// TIA Portal V20 export
DATA_BLOCK "ProcessValues_DB"   // DB34
AUTHOR : Siemens AG
FAMILY : ServiceControl
VERSION : 1.0
// stored: InstanceOfName ProcessValues, InstanceOfType FB
"ProcessValues"
   // VAR_INPUT
   //    ProcessValueOutAnalogIn { ExternalAccessible := 'False'; ExternalVisible := 'False'; ExternalWritable := 'False'} : Array[0..0] of "UDT_MTP_AnaProcessValueOut";
   //    ProcessValueOutDigitalIn { ExternalAccessible := 'False'; ExternalVisible := 'False'; ExternalWritable := 'False'} : Array[0..0] of "UDT_MTP_DIntProcessValueOut";
   //    ProcessValueOutBinaryIn { ExternalAccessible := 'False'; ExternalVisible := 'False'; ExternalWritable := 'False'} : Array[0..0] of "UDT_MTP_BinProcessValueOut";
   //    ProcessValueOutStringIn { ExternalAccessible := 'False'; ExternalVisible := 'False'; ExternalWritable := 'False'} : Array[0..0] of "UDT_MTP_StringProcessValueOut";
   //    ProcessValueInAnalogApply { ExternalAccessible := 'False'; ExternalVisible := 'False'; ExternalWritable := 'False'} : Array[0..0] of "UDT_Service_ProcessValueInApply";
   //    ProcessValueInDigitalApply { ExternalAccessible := 'False'; ExternalVisible := 'False'; ExternalWritable := 'False'} : Array[0..0] of "UDT_Service_ProcessValueInApply";
   // END_VAR
   // VAR_OUTPUT
   //    ProcessValueInAnalogOut { ExternalAccessible := 'False'; ExternalVisible := 'False'; ExternalWritable := 'False'} : Array[0..0] of "UDT_MTP_AnaProcessValueOut";
   //    ProcessValueInDigitalOut { ExternalAccessible := 'False'; ExternalVisible := 'False'; ExternalWritable := 'False'} : Array[0..0] of "UDT_MTP_DIntProcessValueOut";
   //    ProcessValueInBinaryOut { ExternalAccessible := 'False'; ExternalVisible := 'False'; ExternalWritable := 'False'} : Array[0..0] of "UDT_MTP_BinProcessValueOut";
   //    ProcessValueInStringOut { ExternalAccessible := 'False'; ExternalVisible := 'False'; ExternalWritable := 'False'} : Array[0..0] of "UDT_MTP_StringProcessValueOut";
   // END_VAR
   // VAR
   //    MTPAnalogIn : Array[0..4] of "UDT_MTP_AnaProcessValueIn";
   //    MTPDigitalIn : Array[0..0] of "UDT_MTP_DIntProcessValueIn";
   //    MTPBinaryIn : Array[0..0] of "UDT_MTP_BinProcessValueIn";
   //    MTPStringIn : Array[0..0] of "UDT_MTP_StringProcessValueIn";
   //    AnalogIn { ExternalAccessible := 'False'; ExternalVisible := 'False'; ExternalWritable := 'False'; S7_SetPoint := 'True'} : Array[0..0] of "ProcessValueInAnalog";
   //    DigitalIn { ExternalAccessible := 'False'; ExternalVisible := 'False'; ExternalWritable := 'False'; S7_SetPoint := 'True'} : Array[0..0] of "ProcessValueInDigital";
   //    BinaryIn { ExternalAccessible := 'False'; ExternalVisible := 'False'; ExternalWritable := 'False'; S7_SetPoint := 'True'} : Array[0..0] of "ProcessValueInBinary";
   //    StringIn { ExternalAccessible := 'False'; ExternalVisible := 'False'; ExternalWritable := 'False'; S7_SetPoint := 'True'} : Array[0..0] of "ProcessValueInString";
   //    MTPAnalogOut : Array[0..10] of "UDT_MTP_AnaProcessValueOut";
   //    MTPDigitalOut : Array[0..0] of "UDT_MTP_DIntProcessValueOut";
   //    MTPBinaryOut : Array[0..2] of "UDT_MTP_BinProcessValueOut";
   //    MTPStringOut : Array[0..0] of "UDT_MTP_StringProcessValueOut";
   //    AnalogOut { ExternalAccessible := 'False'; ExternalVisible := 'False'; ExternalWritable := 'False'; S7_SetPoint := 'True'} : Array[0..0] of "ProcessValueOutAnalog";
   //    DigitalOut { ExternalAccessible := 'False'; ExternalVisible := 'False'; ExternalWritable := 'False'; S7_SetPoint := 'True'} : Array[0..0] of "ProcessValueOutDigital";
   //    BinaryOut { ExternalAccessible := 'False'; ExternalVisible := 'False'; ExternalWritable := 'False'; S7_SetPoint := 'True'} : Array[0..0] of "ProcessValueOutBinary";
   //    StringOut { ExternalAccessible := 'False'; ExternalVisible := 'False'; ExternalWritable := 'False'; S7_SetPoint := 'True'} : Array[0..0] of "ProcessValueOutString";
   // END_VAR
BEGIN
   MTPAnalogIn[0..2].V := 5.0;
   MTPAnalogIn[3].V := 16.0;
   MTPAnalogIn[0..3].SclMinCur := 0.0;
   MTPAnalogIn[0..2].SclMaxCur := 11.0;
   MTPAnalogIn[3].SclMaxCur := 32.0;
   MTPAnalogIn[0..3].UnitCur := 1351;
   MTPAnalogIn[0..3].SclMinExt := 0.0;
   MTPAnalogIn[0..2].SclMaxExt := 11.0;
   MTPAnalogIn[3].SclMaxExt := 32.0;
   MTPAnalogIn[0..3].UnitExt := 1351;
   MTPAnalogOut[0..10].V := 0.0;
   MTPAnalogOut[0..10].VSclMin := 0.0;
   MTPAnalogOut[0..3].VSclMax := 3000.0;
   MTPAnalogOut[4..7].VSclMax := 100.0;
   MTPAnalogOut[8..9].VSclMax := 3000.0;
   MTPAnalogOut[10].VSclMax := 3200.0;
   MTPAnalogOut[0..3].VUnit := 1038;
   MTPAnalogOut[4..7].VUnit := 1001;
   MTPAnalogOut[8..10].VUnit := 1038;
   MTPBinaryOut[0..1].V := False;
   MTPBinaryOut[0..1].VState0 := 'VlvClosed';
   MTPBinaryOut[0..1].VState1 := 'VlvOpened';
END_DATA_BLOCK
